// TIA Portal V20 export
DATA_BLOCK "InstCallEquipment"   // DB22
{ DB_Accessible_From_OPC_UA := 'FALSE' }
AUTHOR : ERsystem_FA2_DH. Kim
// stored: AssignedProDiagFB Unit1.Em0.ProDiag, DBAccessibleFromOPCUA false, DBAccessibleFromWebserver false, InstanceOfName Unit1.Em0.CallEquipment, InstanceOfType FB, Namespace Unit1.Em0
"Unit1.Em0.CallEquipment"
   // VAR_INPUT
   //    ZoneOperationEnable { ExternalWritable := 'False'} : "LWONIK_typeSafetyZoneManualOperation";
   // END_VAR
   // VAR_IN_OUT
   //    unitStatus : "LAF_typeUnitStatus";
   //    unitAlarmDB : "LAF_typeAlarms";
   //    emFeedback : "LUC_typeEmFeedback";
   // END_VAR
   // VAR
   //    instSequenceUnwinder { S7_SetPoint := 'True'} : "Unit1.Em0.Sequence_1_SepaUnwinderTop";
   //    instTopHomeJob1 { S7_SetPoint := 'True'} : "LAF_SelectJob";
   //    instTopUnwindingJob2 { S7_SetPoint := 'True'} : "LAF_SelectJob";
   //    instTopRewidnigJob10 { S7_SetPoint := 'True'} : "LAF_SelectJob";
   //    instCmTopDirectionCheckSensor { S7_SetPoint := 'True'} : "LBC_DigitalSignalCn";
   //    instCmUnwinderTopRadiusMeasure { ExternalAccessible := 'False'; ExternalVisible := 'False'; ExternalWritable := 'False'} : "LBC_AnalogInputCn";
   //    instCmRadiusMeasure { S7_SetPoint := 'True'} : "LER_RadiusMeasure";
   //    instCmUnwinderTopAxisB { S7_SetPoint := 'True'} : "LBC_Axis64Pos_TecPlcCn";
   //    instInterlockCmUnwinderTopAxisB { S7_SetPoint := 'True'} : "LER_Axis64Pos_InterlockSummary";
   //    instCmUnwinderAirShaftTopOnOff { ExternalAccessible := 'False'; ExternalVisible := 'False'; ExternalWritable := 'False'; S7_SetPoint := 'True'} : "LBC_TwoWayActuatorCn";
   //    instCmUnwinderTopEpcControllerInterface { ExternalAccessible := 'False'; ExternalVisible := 'False'; ExternalWritable := 'False'; S7_SetPoint := 'True'} : "LER_EPC_CON600";
   //    instManageAlarms { ExternalWritable := 'False'} : "LAF_ManageAlarms";
   //    instEventsPFE : "Unit1.Em0.EventsPFE";
   //    instLER_BrakeTestUnwinderTopAxisB : "LER_BrakeTest";
   //    statUnitStatus { ExternalWritable := 'False'} : "LAF_typeUnitStatus";
   //    statSlmStatus : Struct
   //       running { ExternalWritable := 'False'} : Bool;
   //       powerOff { ExternalWritable := 'False'} : Bool;
   //    END_STRUCT;
   //    statAllBrakeTest { ExternalWritable := 'False'} : "LER_typeBrakeTestUnitCommands";
   //    statTonTime { ExternalAccessible := 'False'; ExternalVisible := 'False'; ExternalWritable := 'False'} : Array[0..1999] of TON_TIME;
   //    statTofTime { ExternalAccessible := 'False'; ExternalVisible := 'False'; ExternalWritable := 'False'} : Array[0..99] of TOF_TIME;
   //    statPulse { ExternalAccessible := 'False'; ExternalVisible := 'False'; ExternalWritable := 'False'} : Struct
   //       miscellaneous : Array[0..99] of Bool;
   //       workingDone : Struct
   //          mainPnP : Array[0..99] of Bool;
   //          alignTable : Array[0..99] of Bool;
   //          ngPnP : Array[0..99] of Bool;
   //       END_STRUCT;
   //       axisEnable : Array[0..99] of Bool;
   //       brakeTest : Array[0..99] of Bool;
   //    END_STRUCT;
   //    statEnableManualCmds : Bool := TRUE;
   //    statRcEnableCmds : Bool;
   //    Scan_on { ExternalAccessible := 'False'; ExternalVisible := 'False'; ExternalWritable := 'False'} : Bool;
   //    "*** Interlock Axis ***" { ExternalAccessible := 'False'; ExternalVisible := 'False'; ExternalWritable := 'False'} : Bool;
   //    "UnwinderTopAxisB Home" { S7_SetPoint := 'True'} : "Homing.LER_Axis";
   //    "UnwinderTopAxisB Jog_CW" { S7_SetPoint := 'True'} : "Jog.LER_Axis";
   //    "UnwinderTopAxisB Jog_CCW" { S7_SetPoint := 'True'} : "Jog.LER_Axis";
   //    "UnwinderTopAxisB Position" { S7_SetPoint := 'True'} : Array[0..5] of "Position.LER_Axis";
   //    "*** Interlock Actuator ******" { ExternalAccessible := 'False'; ExternalVisible := 'False'; ExternalWritable := 'False'} : Bool;
   //    "UnwinderAirShaftTop On" { S7_SetPoint := 'True'} : "Cylinder.LER_Actuator";
   //    "UnwinderAirShaftTop Off" { S7_SetPoint := 'True'} : "Cylinder.LER_Actuator";
   //    AXIS1 : "LER_CM_Name";
   //    Cylinder1 : "LER_CM_Name";
   //    citi_Ptrig : Array[0..20] of Bool;
   //    citiTon : Array[0..20] of TON_TIME;
   //    citi : Time;
   //    citiTest : Array[0..20] of Bool;
   // END_VAR
BEGIN
   ZoneOperationEnable.autoStartEnable := FALSE;
   ZoneOperationEnable.doorLockEnable := TRUE;
   ZoneOperationEnable.doorUnlockEnable := TRUE;
   ZoneOperationEnable.rc_AutoEnable := FALSE;
   ZoneOperationEnable.rc_RollChangeEnable := FALSE;
   ZoneOperationEnable.rc_DoorLockEnable := TRUE;
   ZoneOperationEnable.rc_DoorUnlockEnable := TRUE;
   ZoneOperationEnable.hmiOperationEnable := TRUE;
   ZoneOperationEnable.phmiOperationEnable := FALSE;
   instCmTopDirectionCheckSensor.enable := TRUE;
   instCmTopDirectionCheckSensor.parentReferenceDesignator := WSTRING#'U1.EM0 SepaUnwinderTop';
   instCmTopDirectionCheckSensor.digitalValue := FALSE;
   instCmTopDirectionCheckSensor.simulatedDigitalValue := FALSE;
   instCmTopDirectionCheckSensor.statProcessValues.enable := TRUE;
   instCmTopDirectionCheckSensor.statProcessValues.referenceDesignator := WSTRING#'U1.EM0 SepaUnwinderTop.cmTopDirectionCheckSensor';
   instCmTopDirectionCheckSensor.statProcessValues.simulation := FALSE;
   instCmTopDirectionCheckSensor.statProcessValues.processValue := FALSE;
   instCmTopDirectionCheckSensor.statProcessValues.error := FALSE;
   instCmTopDirectionCheckSensor.statProcessValues.status := 16#0000;
   instCmTopDirectionCheckSensor.statDiagnostics.status := 16#0000;
   instCmTopDirectionCheckSensor.statDiagnostics.subfunctionStatus := 16#0000;
   instCmTopDirectionCheckSensor.statDiagnostics.stateNumber := 0;
   instCmTopDirectionCheckSensor.statEmptyDiagnostics.status := 16#0000;
   instCmTopDirectionCheckSensor.statEmptyDiagnostics.subfunctionStatus := 16#0000;
   instCmTopDirectionCheckSensor.statEmptyDiagnostics.stateNumber := 0;
   instCmTopDirectionCheckSensor.instOnDelay.PT := T#0MS;
   instCmTopDirectionCheckSensor.instOnDelay.IN := FALSE;
   instCmTopDirectionCheckSensor.instOffDelay.PT := T#0MS;
   instCmTopDirectionCheckSensor.instOffDelay.IN := FALSE;
   instCmTopDirectionCheckSensor.statDisableAlarms := FALSE;
   instCmTopDirectionCheckSensor.statErrorState := 16#0000;
   instCmTopDirectionCheckSensor.statFirstCall := FALSE;
   instCmTopDirectionCheckSensor.statResetPrevious := FALSE;
   instCmTopDirectionCheckSensor.statEnablePrevious := TRUE;
   instCmTopDirectionCheckSensor.statProcessValuePrevious := FALSE;
   instCmUnwinderTopRadiusMeasure.enable := TRUE;
   instCmUnwinderTopRadiusMeasure.parentReferenceDesignator := WSTRING#'U1.EM0 SepaUnwinderTop';
   instCmUnwinderTopRadiusMeasure.analogValue := -32768;
   instCmUnwinderTopRadiusMeasure.simulatedAnalogValue := 0;
   instCmUnwinderTopRadiusMeasure.statProcessValues.enable := TRUE;
   instCmUnwinderTopRadiusMeasure.statProcessValues.referenceDesignator := WSTRING#'U1.EM0 SepaUnwinderTop.cmTopRadiusMeasure';
   instCmUnwinderTopRadiusMeasure.statProcessValues.simulation := FALSE;
   instCmUnwinderTopRadiusMeasure.statProcessValues.processValue := 0.0;
   instCmUnwinderTopRadiusMeasure.statProcessValues.analogValue := -4864;
   instCmUnwinderTopRadiusMeasure.statProcessValues.limitHigh2 := FALSE;
   instCmUnwinderTopRadiusMeasure.statProcessValues.limitHigh1 := FALSE;
   instCmUnwinderTopRadiusMeasure.statProcessValues.limitLow1 := FALSE;
   instCmUnwinderTopRadiusMeasure.statProcessValues.limitLow2 := FALSE;
   instCmUnwinderTopRadiusMeasure.statProcessValues.maxValueReached := FALSE;
   instCmUnwinderTopRadiusMeasure.statProcessValues.minValueReached := TRUE;
   instCmUnwinderTopRadiusMeasure.statProcessValues.error := TRUE;
   instCmUnwinderTopRadiusMeasure.statProcessValues.status := 16#8405;
   instCmUnwinderTopRadiusMeasure.statDiagnostics.status := 16#8405;
   instCmUnwinderTopRadiusMeasure.statDiagnostics.subfunctionStatus := 16#0000;
   instCmUnwinderTopRadiusMeasure.statDiagnostics.stateNumber := 0;
   instCmUnwinderTopRadiusMeasure.statEmptyDiagnostics.status := 16#0000;
   instCmUnwinderTopRadiusMeasure.statEmptyDiagnostics.subfunctionStatus := 16#0000;
   instCmUnwinderTopRadiusMeasure.statEmptyDiagnostics.stateNumber := 0;
   instCmUnwinderTopRadiusMeasure.statLimitationMessage := '-31.64 mm < 0.00 mm';
   instCmUnwinderTopRadiusMeasure.statLimitMessage := '';
   instCmUnwinderTopRadiusMeasure.statErrorState := 16#8405;
   instCmUnwinderTopRadiusMeasure.statFirstCall := FALSE;
   instCmUnwinderTopRadiusMeasure.statDisableAlarms := TRUE;
   instCmUnwinderTopRadiusMeasure.statResetPrevious := FALSE;
   instCmUnwinderTopRadiusMeasure.statEnablePrevious := TRUE;
   instCmRadiusMeasure.enable := TRUE;
   instCmRadiusMeasure.enableManualCmds := TRUE;
   instCmRadiusMeasure.radiusProcessValue := 0.0;
   instCmRadiusMeasure.radius := 39.0;
   instCmRadiusMeasure.diameter := 78.0;
   instCmRadiusMeasure.statRadiusProcessValueZeroSetOffset := 0.0;
   instCmRadiusMeasure.statRadiusProcessValueBuffer[0] := 0.0;
   instCmRadiusMeasure.statRadiusProcessValueBuffer[1] := 39.0;
   instCmRadiusMeasure.statRadiusProcessValueBuffer[2..3] := 390.0;
   instCmRadiusMeasure.statRadiusProcessValueBuffer[4] := 39.0;
   instCmRadiusMeasure.statRadiusProcessValueBuffer[5] := 0.0;
   instCmRadiusMeasure.statOffset := 0.0;
   instCmUnwinderAirShaftTopOnOff.enable := TRUE;
   instCmUnwinderAirShaftTopOnOff.parentReferenceDesignator := WSTRING#'U1.EM0 SepaUnwinderTop';
   instCmUnwinderAirShaftTopOnOff.feedbackHomePos := FALSE;
   instCmUnwinderAirShaftTopOnOff.feedbackWorkPos := FALSE;
   instCmUnwinderAirShaftTopOnOff.enableManualCmds := TRUE;
   instCmUnwinderAirShaftTopOnOff.interlockWorkPos := TRUE;
   instCmUnwinderAirShaftTopOnOff.interlockHomePos := TRUE;
   instCmUnwinderAirShaftTopOnOff.goToHomePos := FALSE;
   instCmUnwinderAirShaftTopOnOff.goToWorkPos := FALSE;
   instCmUnwinderAirShaftTopOnOff.statProcessValues.enable := TRUE;
   instCmUnwinderAirShaftTopOnOff.statProcessValues.referenceDesignator := WSTRING#'U1.EM0 SepaUnwinderTop.cmAirShaftTopOnOff';
   instCmUnwinderAirShaftTopOnOff.statProcessValues.commandHomePos := FALSE;
   instCmUnwinderAirShaftTopOnOff.statProcessValues.commandWorkPos := FALSE;
   instCmUnwinderAirShaftTopOnOff.statProcessValues.goToHomePos := FALSE;
   instCmUnwinderAirShaftTopOnOff.statProcessValues.goToWorkPos := FALSE;
   instCmUnwinderAirShaftTopOnOff.statProcessValues.inHomePos := FALSE;
   instCmUnwinderAirShaftTopOnOff.statProcessValues.inWorkPos := FALSE;
   instCmUnwinderAirShaftTopOnOff.statProcessValues.reset := FALSE;
   instCmUnwinderAirShaftTopOnOff.statProcessValues.enableManualCmds := TRUE;
   instCmUnwinderAirShaftTopOnOff.statProcessValues.error := FALSE;
   instCmUnwinderAirShaftTopOnOff.statProcessValues.interlockHomePos := TRUE;
   instCmUnwinderAirShaftTopOnOff.statProcessValues.interlockWorkPos := TRUE;
   instCmUnwinderAirShaftTopOnOff.statProcessValues.status := 16#7003;
   instCmUnwinderAirShaftTopOnOff.statProcessValues.interlockWarningWorkPos := FALSE;
   instCmUnwinderAirShaftTopOnOff.statProcessValues.interlockWarningHomePos := FALSE;
   instCmUnwinderAirShaftTopOnOff.statCurrentInputs.commandHomePos := FALSE;
   instCmUnwinderAirShaftTopOnOff.statCurrentInputs.commandWorkPos := FALSE;
   instCmUnwinderAirShaftTopOnOff.statCurrentInputs.reset := FALSE;
   instCmUnwinderAirShaftTopOnOff.statPreviousInputs.commandHomePos := FALSE;
   instCmUnwinderAirShaftTopOnOff.statPreviousInputs.commandWorkPos := FALSE;
   instCmUnwinderAirShaftTopOnOff.statPreviousInputs.reset := FALSE;
   instCmUnwinderAirShaftTopOnOff.statCurrentInterface.commandHomePos := FALSE;
   instCmUnwinderAirShaftTopOnOff.statCurrentInterface.commandWorkPos := FALSE;
   instCmUnwinderAirShaftTopOnOff.statCurrentInterface.reset := FALSE;
   instCmUnwinderAirShaftTopOnOff.statPreviousInterface.commandHomePos := FALSE;
   instCmUnwinderAirShaftTopOnOff.statPreviousInterface.commandWorkPos := FALSE;
   instCmUnwinderAirShaftTopOnOff.statPreviousInterface.reset := FALSE;
   instCmUnwinderAirShaftTopOnOff.statEmptyDiagnostics.status := 16#0000;
   instCmUnwinderAirShaftTopOnOff.statEmptyDiagnostics.subfunctionStatus := 16#0000;
   instCmUnwinderAirShaftTopOnOff.statEmptyDiagnostics.stateNumber := 0;
   instCmUnwinderAirShaftTopOnOff.instTimerReachPos.PT := T#0MS;
   instCmUnwinderAirShaftTopOnOff.instTimerReachPos.IN := FALSE;
   instCmUnwinderAirShaftTopOnOff.instTimerLeavePos.PT := T#0MS;
   instCmUnwinderAirShaftTopOnOff.instTimerLeavePos.IN := FALSE;
   instCmUnwinderAirShaftTopOnOff.instTimerDiscrepancyCheck.PT := T#0MS;
   instCmUnwinderAirShaftTopOnOff.instTimerDiscrepancyCheck.IN := FALSE;
   instCmUnwinderAirShaftTopOnOff.statDisableAlarms := FALSE;
   instCmUnwinderAirShaftTopOnOff.statDiagnostics.status := 16#7003;
   instCmUnwinderAirShaftTopOnOff.statDiagnostics.subfunctionStatus := 16#0000;
   instCmUnwinderAirShaftTopOnOff.statDiagnostics.stateNumber := 0;
   instCmUnwinderAirShaftTopOnOff.statEnablePrevious := TRUE;
   instCmUnwinderAirShaftTopOnOff.statFirstCall := FALSE;
   instCmUnwinderAirShaftTopOnOff.statResetPrevious := FALSE;
   instCmUnwinderAirShaftTopOnOff.statValid := TRUE;
   instCmUnwinderAirShaftTopOnOff.statBusy := TRUE;
   instCmUnwinderAirShaftTopOnOff.statError := FALSE;
   instCmUnwinderAirShaftTopOnOff.statInterlockWorkOff := FALSE;
   instCmUnwinderAirShaftTopOnOff.statInterlockHomeOff := FALSE;
   instCmUnwinderAirShaftTopOnOff.statFbState := 50;
   instCmUnwinderAirShaftTopOnOff.statFbStatePrevious := 50;
   instCmUnwinderAirShaftTopOnOff.statErrorUserCleared := FALSE;
   instCmUnwinderAirShaftTopOnOff.statErrorAutoCleared := FALSE;
   instCmUnwinderAirShaftTopOnOff.statErrorState := 16#0000;
   instCmUnwinderAirShaftTopOnOff.statDisablingCompleted := FALSE;
   instCmUnwinderAirShaftTopOnOff.statFeedbackHomePos := FALSE;
   instCmUnwinderAirShaftTopOnOff.statFeedbackWorkPos := FALSE;
   instManageAlarms.proDiagState.Total_Number := 428;
   instManageAlarms.proDiagState.All := TRUE;
   instManageAlarms.proDiagState.O := FALSE;
   instManageAlarms.proDiagState.I := FALSE;
   instManageAlarms.proDiagState.R := FALSE;
   instManageAlarms.proDiagState."A" := FALSE;
   instManageAlarms.proDiagState.P := FALSE;
   instManageAlarms.proDiagState.Merr := TRUE;
   instManageAlarms.proDiagState.Mtxt := FALSE;
   instManageAlarms.proDiagState.SV_Types := 16#20;
   instManageAlarms.proDiagState.C1 := TRUE;
   instManageAlarms.proDiagState.C2 := FALSE;
   instManageAlarms.proDiagState.C3 := FALSE;
   instManageAlarms.proDiagState.C4 := FALSE;
   instManageAlarms.proDiagState.C5 := FALSE;
   instManageAlarms.proDiagState.C6 := FALSE;
   instManageAlarms.proDiagState.C7 := FALSE;
   instManageAlarms.proDiagState.C8 := FALSE;
   instManageAlarms.proDiagState.Categories := 16#01;
   instManageAlarms.proDiagState.Sub_Cat_1 := 16#0000_0001;
   instManageAlarms.proDiagState.Sub_Cat_2 := 16#0000_0000;
   instManageAlarms.proDiagState.Reserved := 16#00;
   instManageAlarms.parentAlarmDB.error := TRUE;
   instManageAlarms.parentAlarmDB.warning := FALSE;
   instManageAlarms.parentAlarmDB.info := FALSE;
   instManageAlarms.alarmDB.error := TRUE;
   instManageAlarms.alarmDB.warning := FALSE;
   instManageAlarms.alarmDB.info := FALSE;
   instManageAlarms.hmiInterfaceDB.error := TRUE;
   instManageAlarms.hmiInterfaceDB.warning := FALSE;
   instManageAlarms.hmiInterfaceDB.info := FALSE;
   statUnitStatus.acknowledgeActive := FALSE;
   statUnitStatus.alarmsDisabled := FALSE;
   statUnitStatus.simulationActive := FALSE;
   statUnitStatus.safetyReleased := TRUE;
   statUnitStatus.specialFunctions.GaugeRnR1AnodeAlign := FALSE;
   statUnitStatus.specialFunctions.GaugeRnR1CathodeAlign := FALSE;
   statUnitStatus.specialFunctions.GaugeRnR3AnodeAlign := FALSE;
   statUnitStatus.specialFunctions.GaugeRnR3CathodeAlign := FALSE;
   statUnitStatus.specialFunctions.releaseEntry := FALSE;
   statUnitStatus.specialFunctions.dryRun := FALSE;
   statUnitStatus.specialFunctions.ReelCutAnodeUnuse := FALSE;
   statUnitStatus.mode.current := 2;
   statUnitStatus.mode.production := FALSE;
   statUnitStatus.mode.maintenance := TRUE;
   statUnitStatus.mode.manual := FALSE;
   statUnitStatus.mode.sleep := FALSE;
   statUnitStatus.mode.deepsleep := FALSE;
   statUnitStatus.mode.userMode04 := FALSE;
   statUnitStatus.mode.userMode05 := FALSE;
   statUnitStatus.mode.userMode06 := FALSE;
   statUnitStatus.mode.userMode07 := FALSE;
   statUnitStatus.mode.userMode08 := FALSE;
   statUnitStatus.mode.userMode09 := FALSE;
   statUnitStatus.mode.userMode10 := FALSE;
   statUnitStatus.mode.userMode11 := FALSE;
   statUnitStatus.mode.userMode12 := FALSE;
   statUnitStatus.mode.userMode13 := FALSE;
   statUnitStatus.state.current := 2;
   statUnitStatus.state.clearing := FALSE;
   statUnitStatus.state.stopped := TRUE;
   statUnitStatus.state.starting := FALSE;
   statUnitStatus.state.idle := FALSE;
   statUnitStatus.state.suspended := FALSE;
   statUnitStatus.state.execute := FALSE;
   statUnitStatus.state.stopping := FALSE;
   statUnitStatus.state.aborting := FALSE;
   statUnitStatus.state.aborted := FALSE;
   statUnitStatus.state.holding := FALSE;
   statUnitStatus.state.held := FALSE;
   statUnitStatus.state.unholding := FALSE;
   statUnitStatus.state.suspending := FALSE;
   statUnitStatus.state.unsuspending := FALSE;
   statUnitStatus.state.resetting := FALSE;
   statUnitStatus.state.completing := FALSE;
   statUnitStatus.state.complete := FALSE;
END_DATA_BLOCK
